FUNCTION IsStringEqualIgnoreCase : BOOL
VAR_INPUT
	iString1:	STRING;
	iString2:	STRING;
END_VAR

IsStringEqualIgnoreCase := F_ToUCase(iString1) = F_ToUCase(iString2);

END_FUNCTION

(* stored: Version 1.1.0.1, ProductVersion 3.1.4026.18
   POU IsStringEqualIgnoreCase: Id {525c75f4-a936-0302-3ca5-5b19765d4276}, SpecialFunc None *)
